TYPE ST_CM_Base :
(**************************************************************************************
 * 	Application		:	BoxControl Framework
 *	Revision		:	$Revision: 404529 $
 *	Revision date	:	$Date: 2018-04-23 08:21:38 +0200 (Mo., 23 Apr 2018) $
 *	Last changed by	:	$Author: b7bolm $
 *	URL				:	$URL: http://almscdc.swisslog.com/repo/SWPD/Development/BoxControlFramework/20_Release/trunk/01_Software/BCF/BCF/JumpStart/20_Product/10_App/10_Base/10_Lib/01_DUTs/ST_CM_Base.TcDUT $
 *
 *	Purpose			:	Base Structure for Condition monitoring 					
 *
 *
 * ------------------------------------------------------------------------------------
 *	Copyright Swisslog [IP AG], Switzerland. All rights reserved.
 * 
 * ------------------------------------------------------------------------------------
 *	
 * 	Revision History: 
 *
 * 	VERSION			DATE			INITIALS			DESCRIPTION
 *	0.1				01.01.2001		swl					Example
 *
 **************************************************************************************)	
STRUCT
	nCurrentTime 	: ULINT; // Current DC-Time of the PLC-Task
	DAQ				: ST_ITC_DAQ;	/// ITC Message
	GDQ				: ST_ITC_GDQ;	/// ITC Message
	Data			: ARRAY[E_CM_Index.E_BEGIN_VARIABLE+1..E_CM_Index.E_END_VARIABLE-1] OF ST_CM_GeneralData; //Process Data used by Condiition Monitoring Method 
	Settings		: ARRAY[E_CM_Index.E_BEGIN_VARIABLE+1..E_CM_Index.E_END_VARIABLE-1] OF ST_CM_Settings; //Settings Data set by Telegram/User
END_STRUCT
END_TYPE

(* stored: Version 1.1.0.1, ProductVersion 3.1.4022.12
   DUT ST_CM_Base: Id {a497ffe2-91aa-4feb-9528-9bf94155d33e} *)
